(*~
<docu>
	<summary>
			Allows to concat strings using fluent interface. It's similar to C# StringBuilder class
			Usage as follows :
			<code>
				ErrorString := _stringBuilder
					.Clear()
					.Append('Error number: ')
					.Append(INT_TO_STRING(ErrorNumber))
					.Append('. Message: ')
					.Append(ErrorMessage)
					.Append('.')
					.ToString();
			</code>
			
			Inspired by Gerhard Barteling blogpost at https://www.plccoder.com/fluent-code/
	</summary>				
</docu>	
~*)	
FUNCTION_BLOCK StringBuilder
VAR
	{attribute 'hide'}
    _workString:STRING;
END_VAR

METHOD Append : REFERENCE TO StringBuilder
VAR_INPUT
    Text :STRING; 
END_VAR
_workString := Concat(_workString,text);
Append REF= THIS^;
END_METHOD

METHOD Clear : REFERENCE TO StringBuilder
_workString := '';
Clear REF= THIS^;
END_METHOD

METHOD ToString : STRING
ToString := _workString;
END_METHOD

END_FUNCTION_BLOCK

(* stored: Version 1.1.0.1
   POU StringBuilder: Id {1690d5c1-eb92-04b5-39f9-d1d1b7ea958d}, SpecialFunc None
   Method Append: Id {a9cd2d8b-8145-0c23-206c-ae933c3ebe7f}
   Method Clear: Id {0378ca3b-d134-07c2-0629-05b04e8ddb79}
   Method ToString: Id {dd6389b5-b5c9-06d5-0b23-bf4eff042e8b} *)
